FUNCTION "ST10_PartData" : Void
{ S7_Optimized_Access := 'TRUE' }
VERSION : 0.1
   VAR_INPUT
      iSysMode : "RCS_SysComInterface_V1";
   END_VAR

   VAR_TEMP
      idex : Int;
   END_VAR


BEGIN
END_FUNCTION

